TYPE ST_SegmentNumberOut :
STRUCT
END_STRUCT
END_TYPE

(* stored: Version 1.1.0.1
   DUT ST_SegmentNumberOut: Id {276d0801-6252-016b-3a66-9bd2be106cc5} *)
